// TIA Portal project "Factory_io_automated_warehouse_with tia_portal_s7_plc1200_sequential2" (V16)

(* hardware
DEVICE "S7-1200 station_1"  S7-1200 Station
   slot 0: "Rack_0"  S7-1200 Rack  Rack  V1.0
   slot 1: "PLC_1"  CPU 1212C DC/DC/DC  6ES7 212-1AE40-0XB0  V4.4
*)

// ===== PLC "PLC_1"  CPU 1212C DC/DC/DC =====

VAR_GLOBAL   // PLC tag table "Default tag table"
   "At Entery" AT %I0.0 : Bool;
   "At load" AT %I0.1 : Bool;
   "At Left" AT %I0.2 : Bool;
   "At Middle" AT %I0.3 : Bool;
   "At Right" AT %I0.4 : Bool;
   "At Un Loaded" AT %I0.5 : Bool;
   "At Exit" AT %I0.6 : Bool;
   "Moving X" AT %I0.7 : Bool;
   "Moving Z" AT %I1.0 : Bool;
   "Start" AT %I1.1 : Bool;
   "Reset" AT %I1.2 : Bool;
   "Stop" AT %I1.3 : Bool;
   "Emergency Stop" AT %I1.4 : Bool;
   "Auto" AT %I1.5 : Bool;
   "Entery conveyor" AT %Q0.0 : Bool;
   "Load Conveyor" AT %Q0.1 : Bool;
   "Forks Left" AT %Q0.2 : Bool;
   "Forks right" AT %Q0.3 : Bool;
   "Lift" AT %Q0.4 : Bool;
   "Unloaded Conveyor" AT %Q0.5 : Bool;
   "Exit Conveyor" AT %Q0.6 : Bool;
   "Start Light" AT %Q0.7 : Bool;
   "Reset Light" AT %Q1.0 : Bool;
   "Stop Light" AT %Q1.1 : Bool;
   "Target Postion" AT %QD30 : DInt;
   "Manual" AT %I1.6 : Bool;
   "Memory_for_Steps" AT %M0.0 : Bool;
   "Start_FC_one_time" AT %M0.1 : Bool;
   "negative edge for moving z" AT %M0.3 : Bool;
   "Negative edge for moving x" AT %M0.4 : Bool;
   "negative edge for moving x(1)" AT %M0.5 : Bool;
   "negative edge for moving z(1)" AT %M0.6 : Bool;
   "Negative edge for moving z(2)" AT %M0.7 : Bool;
   "Negative edge for moving z(3)" AT %M1.0 : Bool;
   "negative edge for moving x(2)" AT %M1.1 : Bool;
   "negative edge for moving x(3)" AT %M1.2 : Bool;
   "negative edge for moving z(4)" AT %M1.3 : Bool;
   "negative edge for moving z(5)" AT %M1.4 : Bool;
   "negative edge of at load" AT %M1.6 : Bool;
   "producr counter" AT %MD30 : DInt;
END_VAR

DATA_BLOCK "modes"   // DB1
{ S7_Optimized_Access := 'FALSE' }
VERSION : 0.1
   VAR
      "Reset Mode" : Bool;
      "Manual Mode" : Bool;
      "Auto Mode" : Bool;
   END_VAR
BEGIN
END_DATA_BLOCK

DATA_BLOCK "Step_Data"   // DB2
{ S7_Optimized_Access := 'TRUE' }
VERSION : 0.1
   VAR
      Every_thing_AT_home : Bool;
      "Turn on Entery conveyor" : Bool;
      "Turn on Load Conveyor" : Bool;
      "Extend Forks Left" : Bool;
      "Extend Forks right" : Bool;
      Lift : Bool;
      "Turn on Unloaded Conveyor" : Bool;
      "Turn on Exit Conveyor" : Bool;
      "Target Postion" : DInt;
      "Start Light" : Bool;
      "Reset Light" : Bool;
      "Stop Light" : Bool;
   END_VAR
BEGIN
END_DATA_BLOCK

DATA_BLOCK "Steps"   // DB3
{ S7_Optimized_Access := 'TRUE' }
VERSION : 0.1
   VAR
      Current_step : Int;
   END_VAR
BEGIN
END_DATA_BLOCK

// folder: System blocks/Program resources

DATA_BLOCK "IEC_Counter_0_DB"   // DB4
{ S7_Optimized_Access := 'TRUE' }
AUTHOR : Simatic
FAMILY : IEC
NAME : CNTR
VERSION : 1.0
// stored: InstanceOfName IEC_COUNTER
"IEC_COUNTER"
BEGIN
END_DATA_BLOCK

// folder: (top level)

FUNCTION "Operating Mode" : Void   // FC1, LAD
{ S7_Optimized_Access := 'TRUE' }
VERSION : 0.1
   VAR_TEMP   // added for the SCL form of the ladder/FBD networks
      _w1 : Bool;
      _w2 : Bool;
   END_VAR
BEGIN

REGION Network 1
   // manual
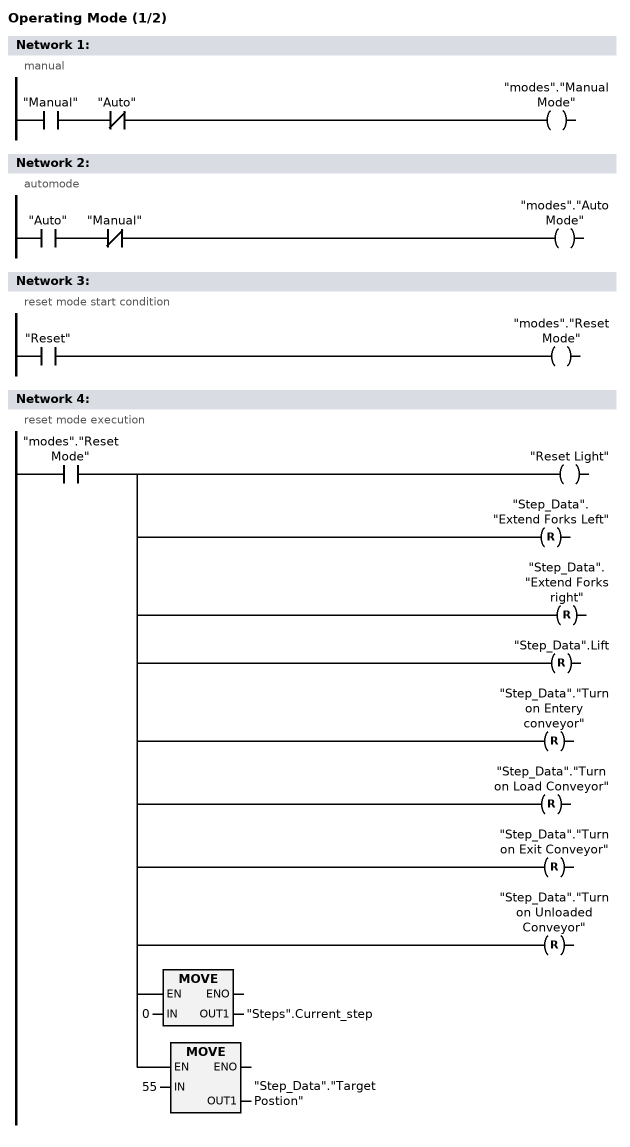
   RUNG wire#powerrail
      Contact( "Manual" )
      I_Contact( "Auto" )
      Coil( "modes"."Manual Mode" )
   END_RUNG
   // the same network as SCL:
   "modes"."Manual Mode" := "Manual" AND NOT "Auto";
END_REGION

REGION Network 2
   // automode
   RUNG wire#powerrail
      Contact( "Auto" )
      I_Contact( "Manual" )
      Coil( "modes"."Auto Mode" )
   END_RUNG
   // the same network as SCL:
   "modes"."Auto Mode" := "Auto" AND NOT "Manual";
END_REGION

REGION Network 3
   // reset mode start condition
   RUNG wire#powerrail
      Contact( "Reset" )
      Coil( "modes"."Reset Mode" )
   END_RUNG
   // the same network as SCL:
   "modes"."Reset Mode" := "Reset";
END_REGION

REGION Network 4
   // reset mode execution
   RUNG wire#powerrail
      Contact( "modes"."Reset Mode" )
      wire#w1
      Coil( "Reset Light" )
   END_RUNG
   RUNG wire#w1
      R_Coil( "Step_Data"."Extend Forks Left" )
   END_RUNG
   RUNG wire#w1
      R_Coil( "Step_Data"."Extend Forks right" )
   END_RUNG
   RUNG wire#w1
      R_Coil( "Step_Data".Lift )
   END_RUNG
   RUNG wire#w1
      R_Coil( "Step_Data"."Turn on Entery conveyor" )
   END_RUNG
   RUNG wire#w1
      R_Coil( "Step_Data"."Turn on Load Conveyor" )
   END_RUNG
   RUNG wire#w1
      R_Coil( "Step_Data"."Turn on Exit Conveyor" )
   END_RUNG
   RUNG wire#w1
      R_Coil( "Step_Data"."Turn on Unloaded Conveyor" )
   END_RUNG
   RUNG wire#w1
      Move(in := 0, out1 => "Steps".Current_step)
   END_RUNG
   RUNG wire#w1
      Move(in := 55, out1 => "Step_Data"."Target Postion")
   END_RUNG
   // the same network as SCL:
   "Reset Light" := "modes"."Reset Mode";
   IF "modes"."Reset Mode" THEN
       "Step_Data"."Extend Forks Left" := FALSE;
       "Step_Data"."Extend Forks right" := FALSE;
       "Step_Data".Lift := FALSE;
       "Step_Data"."Turn on Entery conveyor" := FALSE;
       "Step_Data"."Turn on Load Conveyor" := FALSE;
       "Step_Data"."Turn on Exit Conveyor" := FALSE;
       "Step_Data"."Turn on Unloaded Conveyor" := FALSE;
       "Steps".Current_step := 0;
       "Step_Data"."Target Postion" := 55;
   END_IF;
END_REGION

REGION Network 5
   // one step
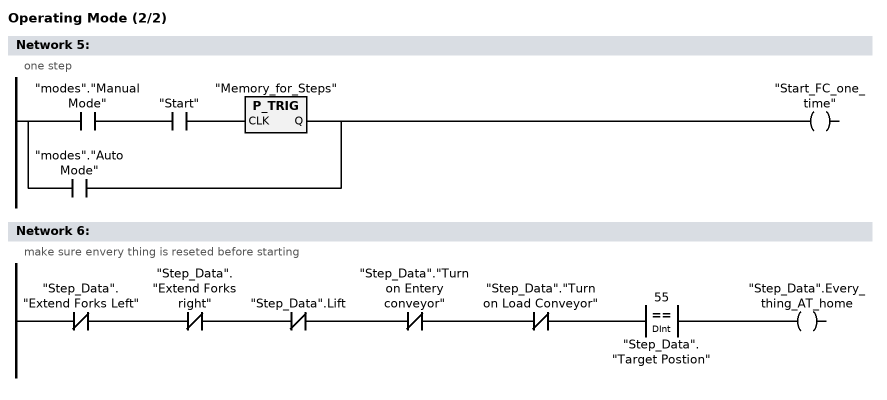
   RUNG wire#powerrail
      Contact( "modes"."Manual Mode" )
      Contact( "Start" )
      P_Trig( "Memory_for_Steps" )
      wire#w1
      Coil( "Start_FC_one_time" )
   END_RUNG
   RUNG wire#powerrail
      Contact( "modes"."Auto Mode" )
   END_RUNG wire#w1
   // the same network as SCL:
   #_w1 := "modes"."Manual Mode" AND "Start";
   #_w2 := #_w1 AND NOT "Memory_for_Steps";   // rising edge
   "Memory_for_Steps" := #_w1;
   "Start_FC_one_time" := #_w2 OR "modes"."Auto Mode";
END_REGION

REGION Network 6
   // make sure envery thing is reseted before starting
   RUNG wire#powerrail
      I_Contact( "Step_Data"."Extend Forks Left" )
      I_Contact( "Step_Data"."Extend Forks right" )
      I_Contact( "Step_Data".Lift )
      I_Contact( "Step_Data"."Turn on Entery conveyor" )
      I_Contact( "Step_Data"."Turn on Load Conveyor" )
      { S7_Templates := "SrcType := DInt" } EQ_Contact(in1 := 55, in2 := "Step_Data"."Target Postion")
      Coil( "Step_Data".Every_thing_AT_home )
   END_RUNG
   // the same network as SCL:
   "Step_Data".Every_thing_AT_home := NOT "Step_Data"."Extend Forks Left" AND NOT "Step_Data"."Extend Forks right" AND NOT "Step_Data".Lift AND NOT "Step_Data"."Turn on Entery conveyor" AND NOT "Step_Data"."Turn on Load Conveyor" AND (55 = "Step_Data"."Target Postion");
END_REGION
END_FUNCTION

FUNCTION "Step_definition" : Void   // FC2, LAD
{ S7_Optimized_Access := 'TRUE' }
VERSION : 0.1
   VAR_TEMP   // added for the SCL form of the ladder/FBD networks
      _w1 : Bool;
      _w2 : Bool;
      _w3 : Bool;
      _w4 : Bool;
   END_VAR
BEGIN

REGION Network 1: trun on load and entery conveyor till negative edge of at load and trun on forks left and counter +1
   // 0---------->1
   // start
   // 8---------->1
   // negative edge of moving z while moving x is off 
   // or negative edge of moving x while moving z is off
   //  or negative edge of moving z and moving x at the same time
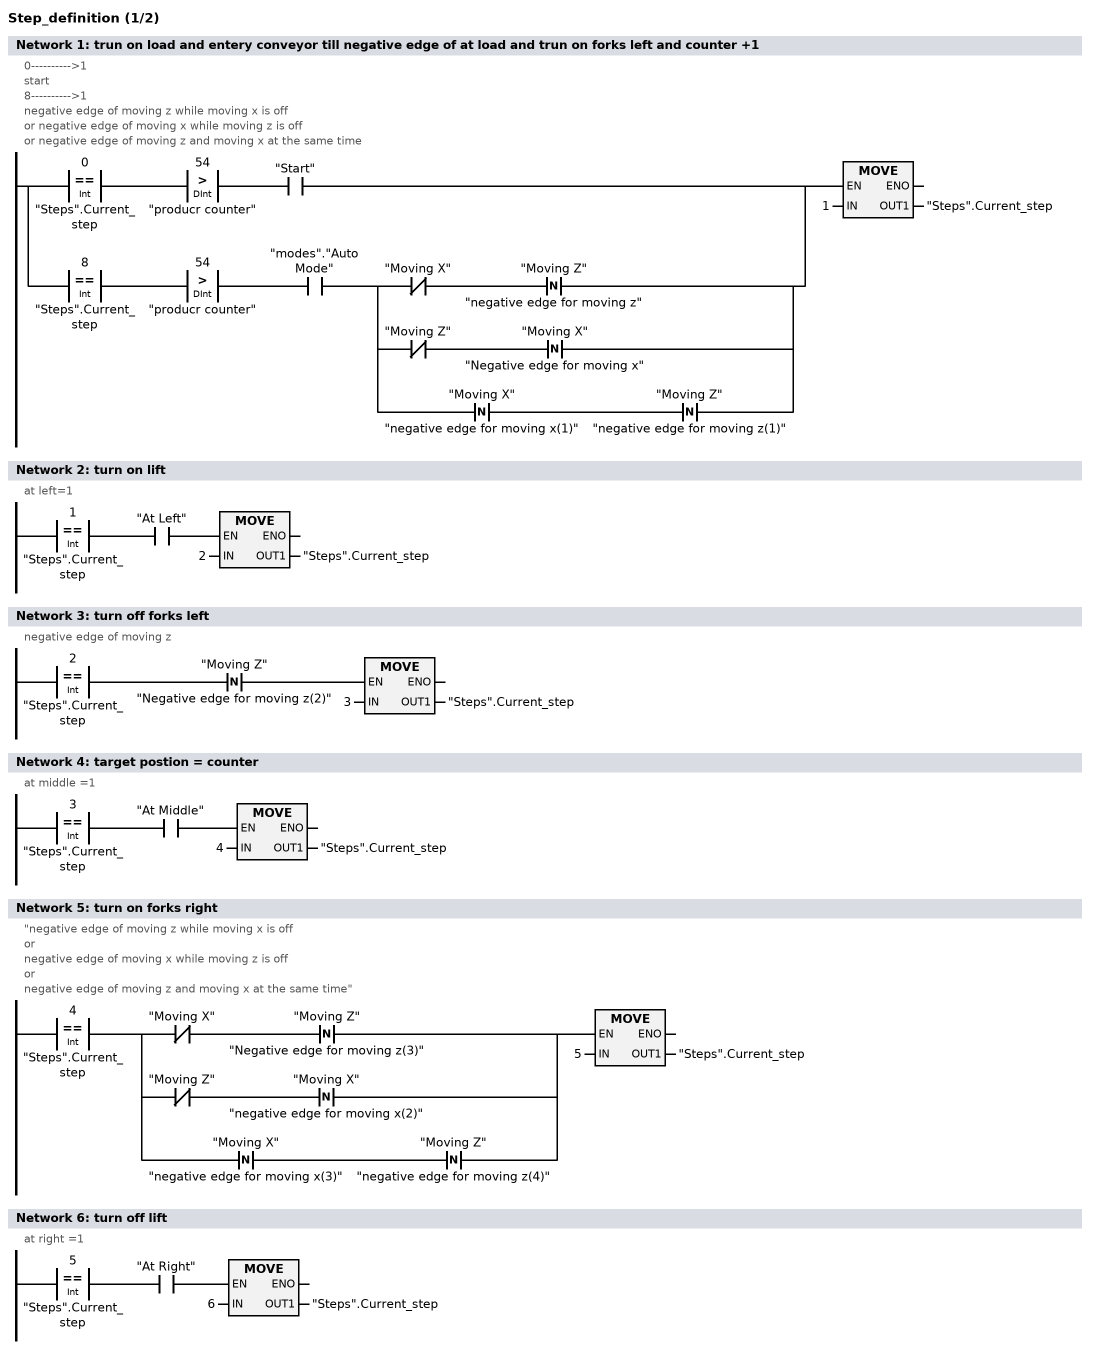
   RUNG wire#powerrail
      { S7_Templates := "SrcType := Int" } EQ_Contact(in1 := 0, in2 := "Steps".Current_step)
      { S7_Templates := "SrcType := DInt" } GT_Contact(in1 := 54, in2 := "producr counter")
      Contact( "Start" )
      wire#w1
      Move(in := 1, out1 => "Steps".Current_step)
   END_RUNG
   RUNG wire#powerrail
      { S7_Templates := "SrcType := Int" } EQ_Contact(in1 := 8, in2 := "Steps".Current_step)
      { S7_Templates := "SrcType := DInt" } GT_Contact(in1 := 54, in2 := "producr counter")
      Contact( "modes"."Auto Mode" )
      wire#w2
      I_Contact( "Moving X" )
      N_Contact(operand := "Moving Z", bit := "negative edge for moving z")
   END_RUNG wire#w1
   RUNG wire#w2
      I_Contact( "Moving Z" )
      N_Contact(operand := "Moving X", bit := "Negative edge for moving x")
   END_RUNG wire#w1
   RUNG wire#w2
      N_Contact(operand := "Moving X", bit := "negative edge for moving x(1)")
      N_Contact(operand := "Moving Z", bit := "negative edge for moving z(1)")
   END_RUNG wire#w1
   // the same network as SCL:
   #_w1 := (8 = "Steps".Current_step) AND (54 > "producr counter") AND "modes"."Auto Mode" AND NOT "Moving X" AND NOT "Moving Z" AND "negative edge for moving z";   // falling edge of "Moving Z"
   "negative edge for moving z" := "Moving Z";
   #_w2 := (8 = "Steps".Current_step) AND (54 > "producr counter") AND "modes"."Auto Mode" AND NOT "Moving Z" AND NOT "Moving X" AND "Negative edge for moving x";   // falling edge of "Moving X"
   "Negative edge for moving x" := "Moving X";
   #_w3 := (8 = "Steps".Current_step) AND (54 > "producr counter") AND "modes"."Auto Mode" AND NOT "Moving X" AND "negative edge for moving x(1)";   // falling edge of "Moving X"
   "negative edge for moving x(1)" := "Moving X";
   #_w4 := #_w3 AND NOT "Moving Z" AND "negative edge for moving z(1)";   // falling edge of "Moving Z"
   "negative edge for moving z(1)" := "Moving Z";
   IF ((0 = "Steps".Current_step) AND (54 > "producr counter") AND "Start") OR #_w1 OR #_w2 OR #_w4 THEN
       "Steps".Current_step := 1;
   END_IF;
END_REGION

REGION Network 2: turn on lift
   // at left=1
   RUNG wire#powerrail
      { S7_Templates := "SrcType := Int" } EQ_Contact(in1 := 1, in2 := "Steps".Current_step)
      Contact( "At Left" )
      Move(in := 2, out1 => "Steps".Current_step)
   END_RUNG
   // the same network as SCL:
   IF (1 = "Steps".Current_step) AND "At Left" THEN "Steps".Current_step := 2; END_IF;
END_REGION

REGION Network 3: turn off forks left
   // negative edge of moving z
   RUNG wire#powerrail
      { S7_Templates := "SrcType := Int" } EQ_Contact(in1 := 2, in2 := "Steps".Current_step)
      N_Contact(operand := "Moving Z", bit := "Negative edge for moving z(2)")
      Move(in := 3, out1 => "Steps".Current_step)
   END_RUNG
   // the same network as SCL:
   #_w1 := (2 = "Steps".Current_step) AND NOT "Moving Z" AND "Negative edge for moving z(2)";   // falling edge of "Moving Z"
   "Negative edge for moving z(2)" := "Moving Z";
   IF #_w1 THEN "Steps".Current_step := 3; END_IF;
END_REGION

REGION Network 4: target postion = counter
   // at middle =1
   RUNG wire#powerrail
      { S7_Templates := "SrcType := Int" } EQ_Contact(in1 := 3, in2 := "Steps".Current_step)
      Contact( "At Middle" )
      Move(in := 4, out1 => "Steps".Current_step)
   END_RUNG
   // the same network as SCL:
   IF (3 = "Steps".Current_step) AND "At Middle" THEN "Steps".Current_step := 4; END_IF;
END_REGION

REGION Network 5: turn on forks right
   // "negative edge of moving z while moving x is off 
   // 
   // or
   //  negative edge of moving x while moving z is off
   // 
   //  or
   //  negative edge of moving z and moving x at the same time"
   RUNG wire#powerrail
      { S7_Templates := "SrcType := Int" } EQ_Contact(in1 := 4, in2 := "Steps".Current_step)
      wire#w1
      I_Contact( "Moving X" )
      N_Contact(operand := "Moving Z", bit := "Negative edge for moving z(3)")
      wire#w2
      Move(in := 5, out1 => "Steps".Current_step)
   END_RUNG
   RUNG wire#w1
      I_Contact( "Moving Z" )
      N_Contact(operand := "Moving X", bit := "negative edge for moving x(2)")
   END_RUNG wire#w2
   RUNG wire#w1
      N_Contact(operand := "Moving X", bit := "negative edge for moving x(3)")
      N_Contact(operand := "Moving Z", bit := "negative edge for moving z(4)")
   END_RUNG wire#w2
   // the same network as SCL:
   #_w1 := (4 = "Steps".Current_step) AND NOT "Moving X" AND NOT "Moving Z" AND "Negative edge for moving z(3)";   // falling edge of "Moving Z"
   "Negative edge for moving z(3)" := "Moving Z";
   #_w2 := (4 = "Steps".Current_step) AND NOT "Moving Z" AND NOT "Moving X" AND "negative edge for moving x(2)";   // falling edge of "Moving X"
   "negative edge for moving x(2)" := "Moving X";
   #_w3 := (4 = "Steps".Current_step) AND NOT "Moving X" AND "negative edge for moving x(3)";   // falling edge of "Moving X"
   "negative edge for moving x(3)" := "Moving X";
   #_w4 := #_w3 AND NOT "Moving Z" AND "negative edge for moving z(4)";   // falling edge of "Moving Z"
   "negative edge for moving z(4)" := "Moving Z";
   IF #_w1 OR #_w2 OR #_w4 THEN "Steps".Current_step := 5; END_IF;
END_REGION

REGION Network 6: turn off lift
   // at right =1
   RUNG wire#powerrail
      { S7_Templates := "SrcType := Int" } EQ_Contact(in1 := 5, in2 := "Steps".Current_step)
      Contact( "At Right" )
      Move(in := 6, out1 => "Steps".Current_step)
   END_RUNG
   // the same network as SCL:
   IF (5 = "Steps".Current_step) AND "At Right" THEN "Steps".Current_step := 6; END_IF;
END_REGION

REGION Network 7: turn off forks right
   // negative edge of moving z
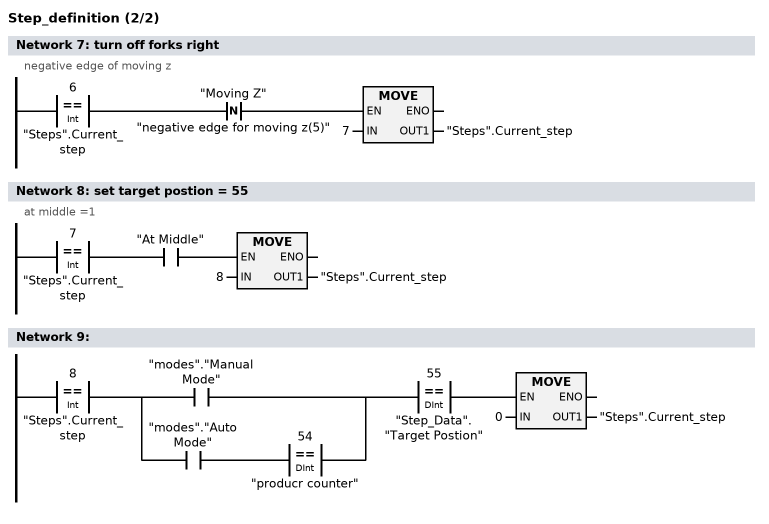
   RUNG wire#powerrail
      { S7_Templates := "SrcType := Int" } EQ_Contact(in1 := 6, in2 := "Steps".Current_step)
      N_Contact(operand := "Moving Z", bit := "negative edge for moving z(5)")
      Move(in := 7, out1 => "Steps".Current_step)
   END_RUNG
   // the same network as SCL:
   #_w1 := (6 = "Steps".Current_step) AND NOT "Moving Z" AND "negative edge for moving z(5)";   // falling edge of "Moving Z"
   "negative edge for moving z(5)" := "Moving Z";
   IF #_w1 THEN "Steps".Current_step := 7; END_IF;
END_REGION

REGION Network 8: set target postion = 55
   // at middle =1
   RUNG wire#powerrail
      { S7_Templates := "SrcType := Int" } EQ_Contact(in1 := 7, in2 := "Steps".Current_step)
      Contact( "At Middle" )
      Move(in := 8, out1 => "Steps".Current_step)
   END_RUNG
   // the same network as SCL:
   IF (7 = "Steps".Current_step) AND "At Middle" THEN "Steps".Current_step := 8; END_IF;
END_REGION

REGION Network 9
   RUNG wire#powerrail
      { S7_Templates := "SrcType := Int" } EQ_Contact(in1 := 8, in2 := "Steps".Current_step)
      wire#w1
      Contact( "modes"."Manual Mode" )
      wire#w2
      { S7_Templates := "SrcType := DInt" } EQ_Contact(in1 := 55, in2 := "Step_Data"."Target Postion")
      Move(in := 0, out1 => "Steps".Current_step)
   END_RUNG
   RUNG wire#w1
      Contact( "modes"."Auto Mode" )
      { S7_Templates := "SrcType := DInt" } EQ_Contact(in1 := 54, in2 := "producr counter")
   END_RUNG wire#w2
   // the same network as SCL:
   IF (8 = "Steps".Current_step) AND ("modes"."Manual Mode" OR ("modes"."Auto Mode" AND (54 = "producr counter"))) AND (55 = "Step_Data"."Target Postion") THEN
       "Steps".Current_step := 0;
   END_IF;
END_REGION
END_FUNCTION

FUNCTION "Step_Execution" : Void   // FC3, LAD
{ S7_Optimized_Access := 'TRUE' }
VERSION : 0.1
   VAR_TEMP   // added for the SCL form of the ladder/FBD networks
      _w1 : Bool;
      _w2 : Bool;
   END_VAR
BEGIN

REGION Network 1: trun on load and entery conveyor till negative edge of at load and trun on forks left and counter +1
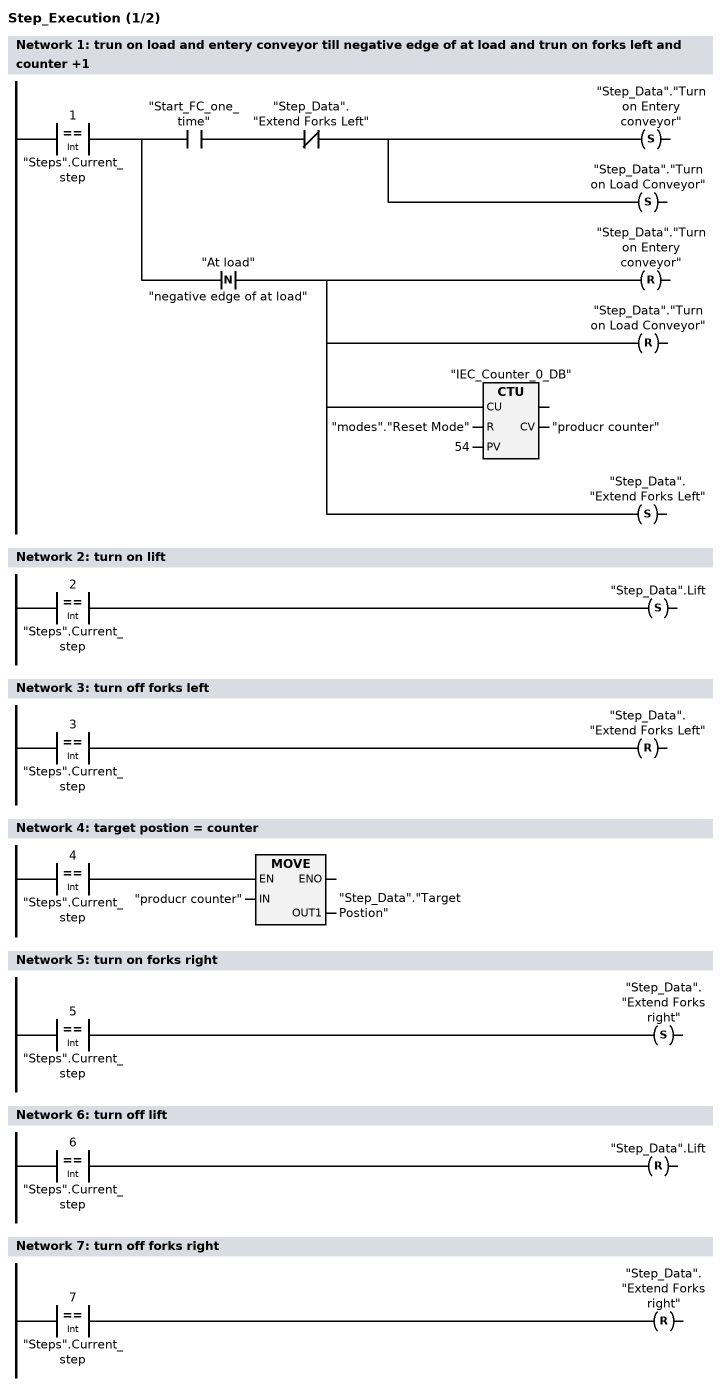
   #_w1 := 1 = "Steps".Current_step;
   IF #_w1 AND "Start_FC_one_time" AND NOT "Step_Data"."Extend Forks Left" THEN
       "Step_Data"."Turn on Entery conveyor" := TRUE;
       "Step_Data"."Turn on Load Conveyor" := TRUE;
   END_IF;
   #_w2 := #_w1 AND NOT "At load" AND "negative edge of at load";   // falling edge of "At load"
   "negative edge of at load" := "At load";
   IF #_w2 THEN
       "Step_Data"."Turn on Entery conveyor" := FALSE;
       "Step_Data"."Turn on Load Conveyor" := FALSE;
   END_IF;
   "IEC_Counter_0_DB".CTU(CU := #_w2, R := "modes"."Reset Mode", PV := 54, CV => "producr counter");
   IF #_w2 THEN "Step_Data"."Extend Forks Left" := TRUE; END_IF;
END_REGION

REGION Network 2: turn on lift
   RUNG wire#powerrail
      { S7_Templates := "SrcType := Int" } EQ_Contact(in1 := 2, in2 := "Steps".Current_step)
      S_Coil( "Step_Data".Lift )
   END_RUNG
   // the same network as SCL:
   IF 2 = "Steps".Current_step THEN "Step_Data".Lift := TRUE; END_IF;
END_REGION

REGION Network 3: turn off forks left
   RUNG wire#powerrail
      { S7_Templates := "SrcType := Int" } EQ_Contact(in1 := 3, in2 := "Steps".Current_step)
      R_Coil( "Step_Data"."Extend Forks Left" )
   END_RUNG
   // the same network as SCL:
   IF 3 = "Steps".Current_step THEN "Step_Data"."Extend Forks Left" := FALSE; END_IF;
END_REGION

REGION Network 4: target postion = counter
   RUNG wire#powerrail
      { S7_Templates := "SrcType := Int" } EQ_Contact(in1 := 4, in2 := "Steps".Current_step)
      Move(in := "producr counter", out1 => "Step_Data"."Target Postion")
   END_RUNG
   // the same network as SCL:
   IF 4 = "Steps".Current_step THEN "Step_Data"."Target Postion" := "producr counter"; END_IF;
END_REGION

REGION Network 5: turn on forks right
   RUNG wire#powerrail
      { S7_Templates := "SrcType := Int" } EQ_Contact(in1 := 5, in2 := "Steps".Current_step)
      S_Coil( "Step_Data"."Extend Forks right" )
   END_RUNG
   // the same network as SCL:
   IF 5 = "Steps".Current_step THEN "Step_Data"."Extend Forks right" := TRUE; END_IF;
END_REGION

REGION Network 6: turn off lift
   RUNG wire#powerrail
      { S7_Templates := "SrcType := Int" } EQ_Contact(in1 := 6, in2 := "Steps".Current_step)
      R_Coil( "Step_Data".Lift )
   END_RUNG
   // the same network as SCL:
   IF 6 = "Steps".Current_step THEN "Step_Data".Lift := FALSE; END_IF;
END_REGION

REGION Network 7: turn off forks right
   RUNG wire#powerrail
      { S7_Templates := "SrcType := Int" } EQ_Contact(in1 := 7, in2 := "Steps".Current_step)
      R_Coil( "Step_Data"."Extend Forks right" )
   END_RUNG
   // the same network as SCL:
   IF 7 = "Steps".Current_step THEN "Step_Data"."Extend Forks right" := FALSE; END_IF;
END_REGION

REGION Network 8
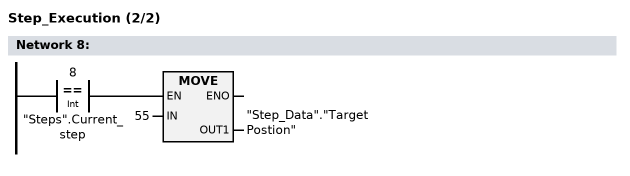
   RUNG wire#powerrail
      { S7_Templates := "SrcType := Int" } EQ_Contact(in1 := 8, in2 := "Steps".Current_step)
      Move(in := 55, out1 => "Step_Data"."Target Postion")
   END_RUNG
   // the same network as SCL:
   IF 8 = "Steps".Current_step THEN "Step_Data"."Target Postion" := 55; END_IF;
END_REGION
END_FUNCTION

FUNCTION "Assignment" : Void   // FC4, LAD
{ S7_Optimized_Access := 'TRUE' }
VERSION : 0.1
BEGIN

REGION Network 1
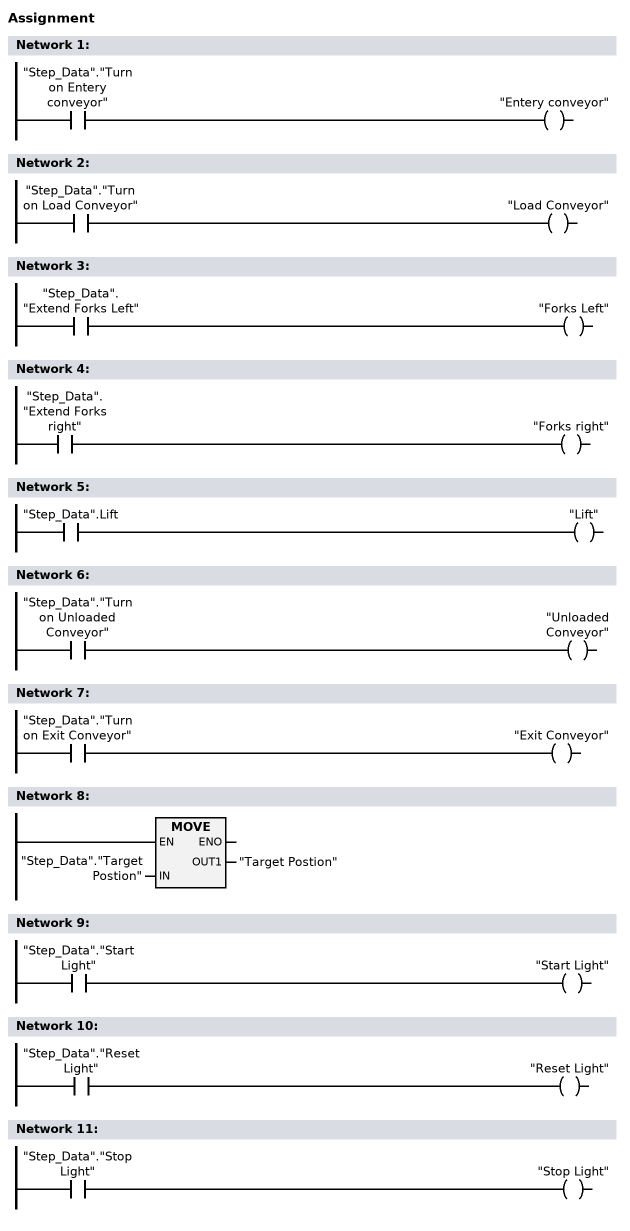
   RUNG wire#powerrail
      Contact( "Step_Data"."Turn on Entery conveyor" )
      Coil( "Entery conveyor" )
   END_RUNG
   // the same network as SCL:
   "Entery conveyor" := "Step_Data"."Turn on Entery conveyor";
END_REGION

REGION Network 2
   RUNG wire#powerrail
      Contact( "Step_Data"."Turn on Load Conveyor" )
      Coil( "Load Conveyor" )
   END_RUNG
   // the same network as SCL:
   "Load Conveyor" := "Step_Data"."Turn on Load Conveyor";
END_REGION

REGION Network 3
   RUNG wire#powerrail
      Contact( "Step_Data"."Extend Forks Left" )
      Coil( "Forks Left" )
   END_RUNG
   // the same network as SCL:
   "Forks Left" := "Step_Data"."Extend Forks Left";
END_REGION

REGION Network 4
   RUNG wire#powerrail
      Contact( "Step_Data"."Extend Forks right" )
      Coil( "Forks right" )
   END_RUNG
   // the same network as SCL:
   "Forks right" := "Step_Data"."Extend Forks right";
END_REGION

REGION Network 5
   RUNG wire#powerrail
      Contact( "Step_Data".Lift )
      Coil( "Lift" )
   END_RUNG
   // the same network as SCL:
   "Lift" := "Step_Data".Lift;
END_REGION

REGION Network 6
   RUNG wire#powerrail
      Contact( "Step_Data"."Turn on Unloaded Conveyor" )
      Coil( "Unloaded Conveyor" )
   END_RUNG
   // the same network as SCL:
   "Unloaded Conveyor" := "Step_Data"."Turn on Unloaded Conveyor";
END_REGION

REGION Network 7
   RUNG wire#powerrail
      Contact( "Step_Data"."Turn on Exit Conveyor" )
      Coil( "Exit Conveyor" )
   END_RUNG
   // the same network as SCL:
   "Exit Conveyor" := "Step_Data"."Turn on Exit Conveyor";
END_REGION

REGION Network 8
   RUNG wire#powerrail
      Move(in := "Step_Data"."Target Postion", out1 => "Target Postion")
   END_RUNG
   // the same network as SCL:
   "Target Postion" := "Step_Data"."Target Postion";
END_REGION

REGION Network 9
   RUNG wire#powerrail
      Contact( "Step_Data"."Start Light" )
      Coil( "Start Light" )
   END_RUNG
   // the same network as SCL:
   "Start Light" := "Step_Data"."Start Light";
END_REGION

REGION Network 10
   RUNG wire#powerrail
      Contact( "Step_Data"."Reset Light" )
      Coil( "Reset Light" )
   END_RUNG
   // the same network as SCL:
   "Reset Light" := "Step_Data"."Reset Light";
END_REGION

REGION Network 11
   RUNG wire#powerrail
      Contact( "Step_Data"."Stop Light" )
      Coil( "Stop Light" )
   END_RUNG
   // the same network as SCL:
   "Stop Light" := "Step_Data"."Stop Light";
END_REGION
END_FUNCTION

FUNCTION "MHJ-PLC-Lab-Function-S71200" : Void   // FC9000, SCL
{ S7_Optimized_Access := 'TRUE' }
VERSION : 0.1
   VAR_TEMP
      rdTimeReturn : Int;
      outputTime : DTL;
      SyncVal : Byte;
      forVal : Int;
      forVal_2 : Int;
      Value : Byte;
   END_VAR
   VAR CONSTANT
      CompVal : Byte := 16#34;
      Value_01 : Byte := 16#11;
      Value_01_DW : DWord := 16#A165_D992;
      Value_02_DW : DWord := 16#58BE_4401;
   END_VAR
BEGIN

   #Value:=PEEK(area := 16#82,
        dbNumber := 0,
        byteOffset := 511);
   #Value := #Value + 1;

   POKE(area := 16#82,
        dbNumber := 0,
        byteOffset := 511,
        value := #Value);

   POKE(area:=16#81,
        dbNumber:=0,
        byteOffset:=1016,
        value:=#Value_01_DW);
   POKE(area := 16#81,
        dbNumber := 0,
        byteOffset := 1020,
        value := #Value_02_DW);

   POKE(area := 16#81,
        dbNumber := 0,
        byteOffset := 511,
        value := B#16#00);

   FOR #forVal := 0 TO 120 DO
       FOR #forVal_2:=0 TO 10 DO
           #rdTimeReturn:=RD_SYS_T(#outputTime);
           #rdTimeReturn := WR_SYS_T(#outputTime);
           #rdTimeReturn := RD_SYS_T(#outputTime);
           #rdTimeReturn := WR_SYS_T(#outputTime);
       END_FOR;
       #SyncVal:= PEEK(area := 16#81,
                      dbNumber := 0,
                      byteOffset := 511);
       IF #SyncVal = #CompVal THEN
          GOTO M_1;
       END_IF;
   END_FOR;
   RETURN;

   M_1:
   POKE(area := 16#81,
        dbNumber := 0,
        byteOffset := 511,
        value := B#16#0);
END_FUNCTION

ORGANIZATION_BLOCK "Main"   // OB1, LAD, ProgramCycle
TITLE = "Main Program Sweep (Cycle)"
{ S7_Optimized_Access := 'TRUE' }
VERSION : 0.1
   VAR_INPUT
      Initial_Call : Bool;   // Initial call of this OB
      Remanence : Bool;   // =True, if remanent data are available
   END_VAR
BEGIN

REGION Network 1
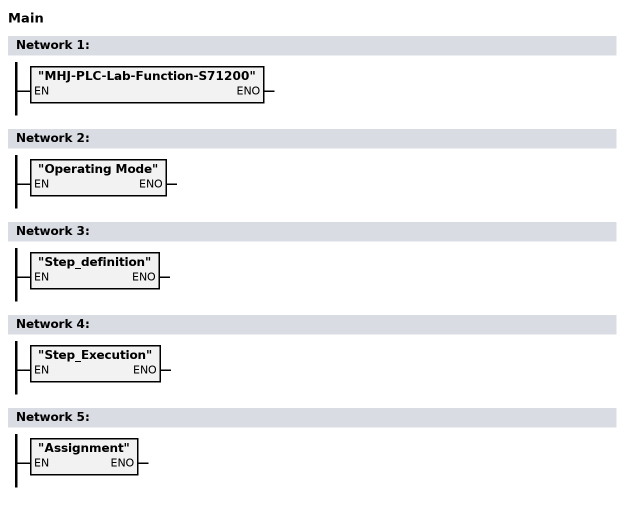
   RUNG wire#powerrail
      "MHJ-PLC-Lab-Function-S71200"()
   END_RUNG
   // the same network as SCL:
   "MHJ-PLC-Lab-Function-S71200"();
END_REGION

REGION Network 2
   RUNG wire#powerrail
      "Operating Mode"()
   END_RUNG
   // the same network as SCL:
   "Operating Mode"();
END_REGION

REGION Network 3
   RUNG wire#powerrail
      "Step_definition"()
   END_RUNG
   // the same network as SCL:
   "Step_definition"();
END_REGION

REGION Network 4
   RUNG wire#powerrail
      "Step_Execution"()
   END_RUNG
   // the same network as SCL:
   "Step_Execution"();
END_REGION

REGION Network 5
   RUNG wire#powerrail
      "Assignment"()
   END_RUNG
   // the same network as SCL:
   "Assignment"();
END_REGION
END_ORGANIZATION_BLOCK